Universal Robots PolyScope program: ProcessFullExperiment.urp

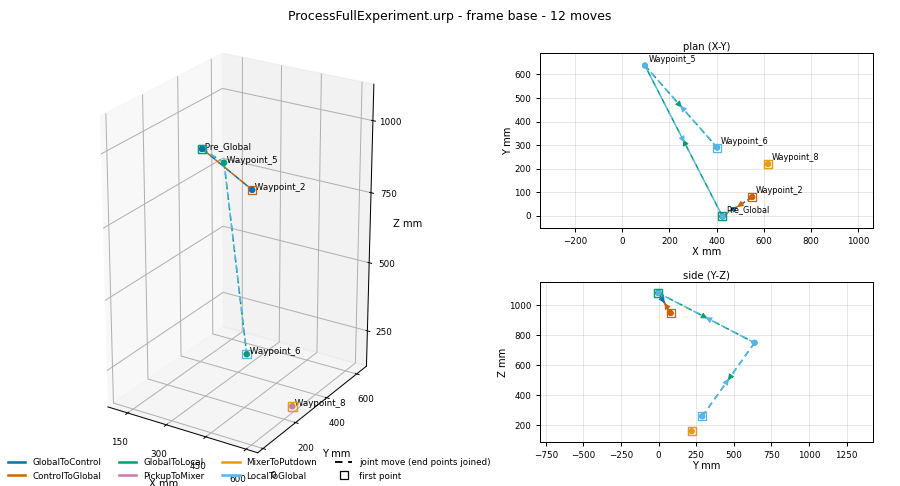
[picture p0: tool path of ProcessFullExperiment.urp in frame base, 12 of 25 moves have a stored position in this frame; points joined in program order, loops and branches not executed]
Program ProcessFullExperiment (installation=Youssef directory=/programs/Youssef createdIn=5.9.5.1031259 lastSavedIn=5.9.5.1031259 robotSerialNumber=20215500597)
Calibrated DH parameters: a=[0.000193, -0.066673, -0.391568, -0.000012, 0.00005, 0]; d=[0.162643, -472.05677, 465.132521, 7.058239, 0.099746, 0.099582]; alpha=[1.571116, 0.00089, 0.003862, 1.569269, -1.569248, 0]; deltaTheta=[0, -1.413394, 7.628392, 0.068187, 0, -0.000001]
Robot Program (runOnlyOnce=true)
  Call ProcessIntensity
  Call ProcessMixing
SubProgram -> ProcessIntensity
SubProgram -> GlobalToControl
SubProgram  [hidden by the author, left out]
SubProgram  [hidden by the author, left out]
SubProgram -> ControlSet
SubProgram  [hidden by the author, left out]
SubProgram  [hidden by the author, left out]
SubProgram  [hidden by the author, left out]
SubProgram  [hidden by the author, left out]
SubProgram  [hidden by the author, left out]
SubProgram  [hidden by the author, left out]
SubProgram -> ControlToGlobal
SubProgram -> ProcessMixing
SubProgram -> GlobalToLocal
SubProgram -> LocalPickup
SubProgram -> PickupToMixer
SubProgram -> MixerToPutdown
SubProgram -> LocalPutdown
SubProgram -> LocalToGlobal
SubProgram ProcessIntensity (keepSynchronizedWithDisk=true) programFile=/programs/Youssef/ProcessIntensity.urp
  Call GlobalToControl
  Call ControlReady
  Call ControlReset
  Call ControlSet
  Call ControlStandby
  Call ControlToGlobal
SubProgram ProcessMixing (keepSynchronizedWithDisk=true) programFile=/programs/Youssef/ProcessMixing.urp
  Call GlobalToLocal
  Call LocalPickup
  Call PickupToMixer
  Wait Sleep waitTime=5
  Call MixerToPutdown
  Call LocalPutdown
  Call LocalToGlobal
SubProgram GlobalToControl (keepSynchronizedWithDisk=true) programFile=/programs/Youssef/GlobalToControl.urp
  MoveJ speed 60 deg/s, acceleration 80 deg/s^2 (useActiveTCP=true) feature=Base
    SafeHome (positionOptionType=SPEED_AND_ACCELERATION speed=1.047198 acceleration=1.396263 nextMotionTime=2)
    Waypoint Pre_Global: TCP in base x=424.817 y=-1.551 z=1080.554 mm, rx=-1.2067 ry=1.2116 rz=-1.2125 rad; joints [89.999, -90, 0, -89.996, -0.001, -0.002] deg; TCP offset x=0 y=0 z=191.5 mm, rx=0 ry=0 rz=0 rad
    URCap Gripper Activate (Robotiq_Grippers, Robotiq Inc.) dataModel(ResetAndActivateKey=false)
    URCap Gripper (Robotiq_Grippers, Robotiq Inc.) dataModel(position=100.0, force=0.0, speed=30.0, positionInDouble=100.0, forceInDouble=0.0, speedInDouble=30.0, slaveIds=[9], blocking=true)
    Waypoint Waypoint_2: TCP in base x=551.14 y=80.155 z=946.388 mm, rx=-1.3882 ry=1.5372 rz=-1.1084 rad; joints [175.158, -73.344, -0.017, -87.688, -91.199, -0.001] deg
    Waypoint Waypoint (Variable): variable(featureName=Control_Standby)
SubProgram ControlReady [hidden by the author, left out]
SubProgram ControlReset [hidden by the author, left out]
SubProgram ControlSet (keepSynchronizedWithDisk=true) programFile=/programs/Youssef/ControlSet.urp
  If GP_int_in[6]≟5
    Call ControlSet5
  ElseIf GP_int_in[6]≟4
    Call ControlSet4
  ElseIf GP_int_in[6]≟3
    Call ControlSet3
  ElseIf GP_int_in[6]≟2
    Call ControlSet2
  Else 
    Call ControlSet1
SubProgram ControlStandby [hidden by the author, left out]
SubProgram ControlToGlobal (keepSynchronizedWithDisk=true) programFile=/programs/Youssef/ControlToGlobal.urp
  MoveJ speed 60 deg/s, acceleration 80 deg/s^2 (useActiveTCP=true) feature=Base
    Waypoint Waypoint (Variable): variable(featureName=Control_Standby)
    Waypoint Waypoint_11: TCP in base x=551.14 y=80.155 z=946.388 mm, rx=-1.3882 ry=1.5372 rz=-1.1084 rad; joints [175.158, -73.344, -0.017, -87.688, -91.199, -0.001] deg
    URCap Gripper (Robotiq_Grippers, Robotiq Inc.) dataModel(position=0.0, force=0.0, speed=30.0, positionInDouble=0.0, forceInDouble=0.0, speedInDouble=30.0, slaveIds=[9], blocking=true)
    URCap Gripper Activate (Robotiq_Grippers, Robotiq Inc.) dataModel(ResetAndActivateKey=false)
    Waypoint Pre_Global_1: TCP in base x=424.817 y=-1.551 z=1080.554 mm, rx=-1.2067 ry=1.2116 rz=-1.2125 rad; joints [89.999, -90, 0, -89.996, -0.001, -0.002] deg
    SafeHome (positionOptionType=SPEED_AND_ACCELERATION speed=1.047198 acceleration=1.396263 nextMotionTime=2)
SubProgram GlobalToLocal (keepSynchronizedWithDisk=true) programFile=/programs/Youssef/GlobalToLocal.urp
  MoveJ speed 60 deg/s, acceleration 80 deg/s^2 (useActiveTCP=true) feature=Base
    SafeHome (positionOptionType=SPEED_AND_ACCELERATION speed=1.047198 acceleration=1.396263 nextMotionTime=2)
    Waypoint Pre_Global_2: TCP in base x=424.817 y=-1.551 z=1080.554 mm, rx=-1.2067 ry=1.2116 rz=-1.2125 rad; joints [89.999, -90, 0, -89.996, -0.001, -0.002] deg
    Waypoint Waypoint_5: TCP in base x=96.27 y=637.775 z=749.236 mm, rx=-1.4855 ry=-0.0307 rz=0.0319 rad; joints [94.292, -84.133, -90.199, -0.883, 88.027, -0.054] deg
    Waypoint Waypoint_6: TCP in base x=402.516 y=290.095 z=259.958 mm, rx=1.3002 ry=1.1489 rz=1.2399 rad; joints [94.435, -83.523, -131.099, -136.444, 6.698, -3.896] deg
    Waypoint Waypoint (Variable): variable(featureName=Local)
SubProgram LocalPickup (keepSynchronizedWithDisk=true) programFile=/programs/Youssef/LocalPickup.urp
  MoveJ speed 60 deg/s, acceleration 80 deg/s^2 (useActiveTCP=true) feature=Base
    Waypoint Waypoint (Variable): variable(featureName=Local)
  URCap Gripper Activate (Robotiq_Grippers, Robotiq Inc.) dataModel(ResetAndActivateKey=false)
  URCap Gripper (Robotiq_Grippers, Robotiq Inc.) dataModel(position=0.0, force=20.0, speed=49.80392156862745, positionInDouble=0.0, forceInDouble=20.0, speedInDouble=49.80392156862745, slaveIds=[9], blocking=true)
  MoveJ speed 60 deg/s, acceleration 80 deg/s^2 (useActiveTCP=true) feature=Base
    Waypoint Waypoint (Variable): variable(featureName=Pickup)
    URCap Gripper (Robotiq_Grippers, Robotiq Inc.) dataModel(position=100.0, force=20.0, speed=50.0, positionInDouble=100.0, forceInDouble=20.0, speedInDouble=50.0, slaveIds=[9], blocking=true)
SubProgram PickupToMixer (keepSynchronizedWithDisk=true) programFile=/programs/Youssef/PickupToMixer.urp
  MoveJ speed 60 deg/s, acceleration 80 deg/s^2 (useActiveTCP=true) feature=Base
    Waypoint Waypoint (Variable): variable(featureName=Pickup)
    URCap Gripper (Robotiq_Grippers, Robotiq Inc.) dataModel(position=100.0, force=49.80392156862745, speed=20.0, positionInDouble=100.0, forceInDouble=49.80392156862745, speedInDouble=20.0, slaveIds=[9], blocking=true)
    Waypoint Waypoint_8: TCP in base x=618.275 y=219.993 z=160.974 mm, rx=1.209 ry=1.2027 rz=1.1964 rad; joints [54.155, -107.639, -124.058, -128.368, -34.984, -0.179] deg
  MoveJ speed 60 deg/s, acceleration 80 deg/s^2 (useActiveTCP=true) feature=Base
    Waypoint Waypoint (Variable): variable(featureName=Mixer_Standby)
    Waypoint Waypoint (Variable): variable(featureName=Mixer_Intact)
SubProgram MixerToPutdown (keepSynchronizedWithDisk=true) programFile=/programs/Youssef/MixerToPutdown.urp
  URCap Gripper (Robotiq_Grippers, Robotiq Inc.) dataModel(position=100.0, force=49.80392156862745, speed=20.0, positionInDouble=100.0, forceInDouble=49.80392156862745, speedInDouble=20.0, slaveIds=[9], blocking=true)
  MoveJ speed 60 deg/s, acceleration 80 deg/s^2 (useActiveTCP=true) feature=Base
    Waypoint Waypoint (Variable): variable(featureName=Mixer_Intact)
    Waypoint Waypoint (Variable): variable(featureName=Mixer_Standby)
  MoveJ speed 60 deg/s, acceleration 80 deg/s^2 (useActiveTCP=true) feature=Base
    Waypoint Waypoint_9: TCP in base x=618.275 y=219.993 z=160.974 mm, rx=1.209 ry=1.2027 rz=1.1964 rad; joints [54.155, -107.639, -124.058, -128.368, -34.984, -0.179] deg
    Waypoint Waypoint (Variable): variable(featureName=Pickup)
    URCap Gripper (Robotiq_Grippers, Robotiq Inc.) dataModel(position=0.0, force=49.80392156862745, speed=20.0, positionInDouble=0.0, forceInDouble=49.80392156862745, speedInDouble=20.0, slaveIds=[9], blocking=true)
SubProgram LocalPutdown (keepSynchronizedWithDisk=true) programFile=/programs/Youssef/LocalPutdown.urp
  URCap Gripper (Robotiq_Grippers, Robotiq Inc.) dataModel(position=0.0, force=20.0, speed=50.0, positionInDouble=0.0, forceInDouble=20.0, speedInDouble=50.0, slaveIds=[9], blocking=true)
  MoveJ speed 60 deg/s, acceleration 80 deg/s^2 (useActiveTCP=true) feature=Base
    Waypoint Waypoint (Variable): variable(featureName=Local)
SubProgram LocalToGlobal (keepSynchronizedWithDisk=true) programFile=/programs/Youssef/LocalToGlobal.urp
  MoveJ speed 60 deg/s, acceleration 80 deg/s^2 (useActiveTCP=true) feature=Base
    Waypoint Waypoint (Variable): variable(featureName=Local)
    Waypoint Waypoint_7: TCP in base x=402.516 y=290.095 z=259.958 mm, rx=1.3002 ry=1.1489 rz=1.2399 rad; joints [94.435, -83.523, -131.099, -136.444, 6.698, -3.896] deg
    Waypoint Waypoint_10: TCP in base x=96.27 y=637.775 z=749.236 mm, rx=-1.4855 ry=-0.0307 rz=0.0319 rad; joints [94.292, -84.133, -90.199, -0.883, 88.027, -0.054] deg
    Waypoint Pre_Global_3: TCP in base x=424.817 y=-1.551 z=1080.554 mm, rx=-1.2067 ry=1.2116 rz=-1.2125 rad; joints [89.999, -90, 0, -89.996, -0.001, -0.002] deg
    SafeHome (positionOptionType=SPEED_AND_ACCELERATION speed=1.047198 acceleration=1.396263 nextMotionTime=2)
SubProgram ControlSet5 [hidden by the author, left out]
SubProgram ControlSet4 [hidden by the author, left out]
SubProgram ControlSet3 [hidden by the author, left out]
SubProgram ControlSet2 [hidden by the author, left out]
SubProgram ControlSet1 [hidden by the author, left out]
